TYPE ST_IOMappingJson :
STRUCT
	name : STRING;
	deviceNum : WORD;
	channel : USINT;
	ethercatDeviceNum : WORD;
	ioLinkDevice : USINT;
	ioLinkSlaveChannel : USINT;	
	pAny : MPM_JsonParser.ST_AnyType_User;
END_STRUCT
END_TYPE

(* stored: Version 1.1.0.1, ProductVersion 3.1.4024.12
   DUT ST_IOMappingJson: Id {ef853e0e-dd6f-4d2c-9889-58888954195a} *)
